PROGRAM MAIN
VAR
	fbMover				: MC_PlanarMover;
	fbM1_Axis			: ARRAY [1..6] OF AXIS_REF;
	iMode				: INT;
END_VAR

GVL.g_fbTcJoy();

CASE iMode OF
	0: 
	ControllerMode(
		fbMover:= fbMover, 
		fbMover_Axis:= fbM1_Axis);
END_CASE

fbMover.Update();

END_PROGRAM

(* stored: Version 1.1.0.1, ProductVersion 3.1.4024.12
   POU MAIN: Id {50777646-4133-4dff-9c0d-35adc043d3ce}, SpecialFunc None *)
